SYSTEM TestMergeFB
  (* Version 1.0, 2023-09-26, ADMIN *)
  APPLICATION TestSampleApp
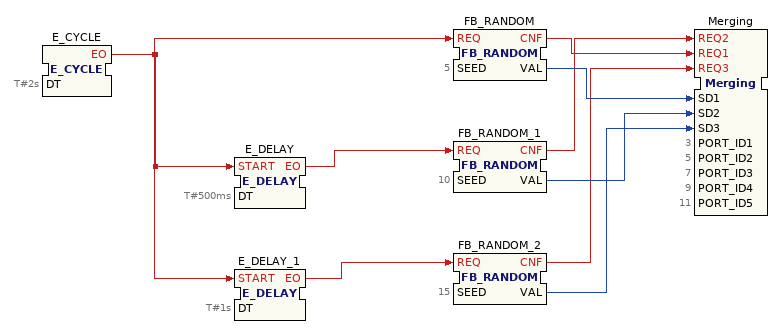
    FBS
      Merging : Merging(PORT_ID1 := 3, PORT_ID2 := 5, PORT_ID3 := 7, PORT_ID4 := 9, PORT_ID5 := 11);
      E_CYCLE : E_CYCLE(DT := T#2s);
      E_DELAY : E_DELAY(DT := T#500ms);
      E_DELAY_1 : E_DELAY(DT := T#1s);
      FB_RANDOM : FB_RANDOM(SEED := 5);
      FB_RANDOM_1 : FB_RANDOM(SEED := 10);
      FB_RANDOM_2 : FB_RANDOM(SEED := 15);
    END_FBS
    EVENT_CONNECTIONS
      E_CYCLE.EO TO E_DELAY.START;
      E_CYCLE.EO TO E_DELAY_1.START;
      E_DELAY.EO TO FB_RANDOM_1.REQ;
      E_DELAY_1.EO TO FB_RANDOM_2.REQ;
      E_CYCLE.EO TO FB_RANDOM.REQ;
      FB_RANDOM_1.CNF TO Merging.REQ2;
      FB_RANDOM.CNF TO Merging.REQ1;
      FB_RANDOM_2.CNF TO Merging.REQ3;
    END_CONNECTIONS
    DATA_CONNECTIONS
      FB_RANDOM.VAL TO Merging.SD1;
      FB_RANDOM_1.VAL TO Merging.SD2;
      FB_RANDOM_2.VAL TO Merging.SD3;
    END_CONNECTIONS
  END_APPLICATION
  DEVICE BeagleBoneBlack : BeagleBoneBlack(MGR_ID := "192.168.7.2:61499")
    {SET_ATTRIBUTE(Profile, HOLOBLOC)} (* device profile *)
    RESOURCE EMB_RES : EMB_RES
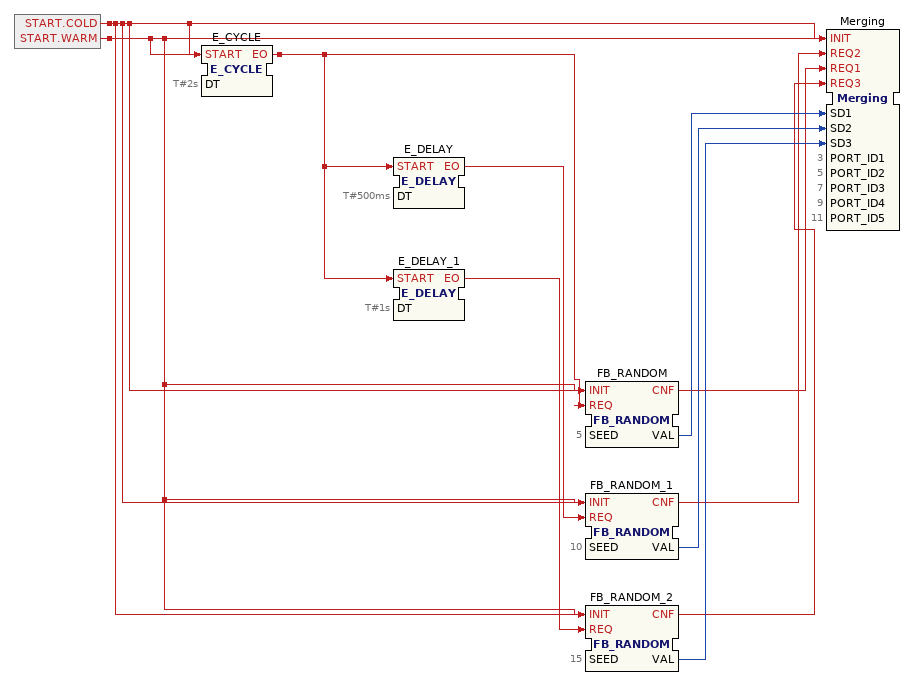
      FBS
        FB_RANDOM_2 : FB_RANDOM(SEED := 15);
        FB_RANDOM_1 : FB_RANDOM(SEED := 10);
        FB_RANDOM : FB_RANDOM(SEED := 5);
        E_DELAY_1 : E_DELAY(DT := T#1s);
        E_DELAY : E_DELAY(DT := T#500ms);
        E_CYCLE : E_CYCLE(DT := T#2s);
        Merging : Merging(PORT_ID1 := 3, PORT_ID2 := 5, PORT_ID3 := 7, PORT_ID4 := 9, PORT_ID5 := 11);
      END_FBS
      EVENT_CONNECTIONS
        START.COLD TO FB_RANDOM_2.INIT;
        START.COLD TO FB_RANDOM_1.INIT;
        START.COLD TO FB_RANDOM.INIT;
        E_CYCLE.EO TO E_DELAY_1.START;
        E_CYCLE.EO TO E_DELAY.START;
        START.WARM TO E_CYCLE.START;
        START.COLD TO E_CYCLE.START;
        START.WARM TO Merging.INIT;
        START.COLD TO Merging.INIT;
        START.WARM TO FB_RANDOM.INIT;
        START.WARM TO FB_RANDOM_1.INIT;
        START.WARM TO FB_RANDOM_2.INIT;
        E_DELAY.EO TO FB_RANDOM_1.REQ;
        E_DELAY_1.EO TO FB_RANDOM_2.REQ;
        E_CYCLE.EO TO FB_RANDOM.REQ;
        FB_RANDOM_1.CNF TO Merging.REQ2;
        FB_RANDOM.CNF TO Merging.REQ1;
        FB_RANDOM_2.CNF TO Merging.REQ3;
      END_CONNECTIONS
      DATA_CONNECTIONS
        FB_RANDOM.VAL TO Merging.SD1;
        FB_RANDOM_1.VAL TO Merging.SD2;
        FB_RANDOM_2.VAL TO Merging.SD3;
      END_CONNECTIONS
    END_RESOURCE
  END_DEVICE
  MAPPINGS
    TestSampleApp.FB_RANDOM_2 ON BeagleBoneBlack.EMB_RES.FB_RANDOM_2;
    TestSampleApp.FB_RANDOM_1 ON BeagleBoneBlack.EMB_RES.FB_RANDOM_1;
    TestSampleApp.FB_RANDOM ON BeagleBoneBlack.EMB_RES.FB_RANDOM;
    TestSampleApp.E_DELAY_1 ON BeagleBoneBlack.EMB_RES.E_DELAY_1;
    TestSampleApp.E_DELAY ON BeagleBoneBlack.EMB_RES.E_DELAY;
    TestSampleApp.E_CYCLE ON BeagleBoneBlack.EMB_RES.E_CYCLE;
    TestSampleApp.Merging ON BeagleBoneBlack.EMB_RES.Merging;
  END_MAPPINGS
  SEGMENTS
    Ethernet : Ethernet;
  END_SEGMENTS
  LINKS
    BeagleBoneBlack => Ethernet;
  END_LINKS
END_SYSTEM
